(* IEC 61131-3 sources: Industry-PLC-LLM/data/PLCBEAD_repo/PLCBEAD_PLCEmbed-main/PLC-BEAD/Source/GEB/SINC, 1 file *)

(* ---- SINC.ST ---- *)
FUNCTION SINC:REAL

	VAR_INPUT
		X :	REAL;
	END_VAR

	IF X = 0.0 THEN
		SINC := 1.0;
	ELSE
		SINC := SIN(X) / x;
	END_IF;

END_FUNCTION

PROGRAM program0

	VAR
		X :	REAL;
		CEIL5_OUT : REAL;
	END_VAR

  	CEIL5_OUT := SINC(X);

END_PROGRAM
